// TIA Portal V18 export
TYPE "ATEQRecipe"
// stored: IsFailsafeCompliant false
   STRUCT
      RessureCurrentValueUL : Real;   // 压力值上限
      RessureCurrentValueLL : Real;   // 压力值下限
      LeakCurrentValueUL : Real;   // 泄露压力值上限
      LeakCurrentValueLL : Real;   // 泄露压力值下限
      PositivePressureProgNo : Int;   // 正压程序号
      NegativePressureProgNo : Int;   // 负压程序号
   END_STRUCT;
END_TYPE
